PROGRAM MAIN_simu
VAR
    simIO : MNG_Simulation;
END_VAR

// Update IOs with simulation
simIO(bEnable := TRUE);

// Application code follows here:

END_PROGRAM

(* stored: Version 1.1.0.1, ProductVersion 3.1.0.25
   POU MAIN_simu: Id {c5c15e1d-44a8-4c3e-a819-f418c54a29eb} *)
